// TwinCAT 3 PLC project PLC_Template
// ProgramVersion: 3.1.4024.0
// libraries:
//   Tc2_Standard, * (Beckhoff Automation GmbH)
//   Tc2_System, * (Beckhoff Automation GmbH)
//   Tc3_Module, * (Beckhoff Automation GmbH)
// project tree:
//   / PlcTask.TcTTO
//   POUs/ MAIN.TcPOU
// real-time tasks:
//   TASK PlcTask: cycle T#10ms, priority 20, ADS port 350
// I/O:
//   DEVICE Device 4 (EtherCAT), AmsNetId 10.110.168.240.5.1
//     Box 1 (DPort-ECT) [DPort-ECT]
// variable links:
//   PLC_Template/PLC_Template Instance <-> Device 4 (EtherCAT)/Box 1 (DPort-ECT)
//     PlcTask Outputs/MAIN.LED_OUT <-> PDOChannel process data mapping/LED1

CONFIGURATION PLC_Template
    RESOURCE PLC ON TwinCAT3
        TASK PlcTask(INTERVAL := T#10ms, PRIORITY := 20);
        PROGRAM MAIN WITH PlcTask : MAIN;
    END_RESOURCE
END_CONFIGURATION

// ---- POUs/MAIN.TcPOU
// 定义程序结构
PROGRAM MAIN
VAR
    TimerOn : TON; // 定时器，用于控制LED亮3秒
    TimerOff : TON; // 定时器，用于控制LED灭3秒
    LED : BOOL := FALSE; // LED状态变量，初始为关闭
	LED_OUT AT %Q*: USINT;
	OnTime : TIME := T#500MS; // LED亮的时间，设置为3秒
    OffTime : TIME := T#500MS; // LED灭的时间，设置为3秒
END_VAR

// 程序逻辑
// 控制LED亮3秒
TimerOn(IN := LED AND NOT TimerOn.Q, PT := OnTime); // 当LED为TRUE且TimerOn未完成时启动
IF TimerOn.Q THEN
    LED := FALSE; // 当TimerOn完成时，切换LED状态为FALSE
END_IF;

// 控制LED灭3秒
TimerOff(IN := NOT LED AND NOT TimerOff.Q, PT := OffTime); // 当LED为FALSE且TimerOff未完成时启动
IF TimerOff.Q THEN
    LED := TRUE; // 当TimerOff完成时，切换LED状态为TRUE
END_IF;

// 根据LED状态设置LED_OUT的值
IF LED THEN
    LED_OUT := 1;   // LED亮
ELSE 
    LED_OUT := 0;   // LED灭
END_IF

END_PROGRAM
